# EPICS alarm handler configuration: mps_database/bareTest/alarms/areas/mpln_bpn19_mp01.alhConfig
GROUP NULL MPLN:BPN19:MP01:1
$ALIAS MPS Link Node 83
$GUIDANCE
LTUH MPS
   Group Name: MPLN:BPN19:MP01:1
   Summary PV:  MPLN:BPN19:MP01:1:STATSUMY
$END
CHANNEL  MPLN:BPN19:MP01:1    MPLN:BPN19:MP01:1:MPS_EN_RBV		-----
CHANNEL  MPLN:BPN19:MP01:1    MPLN:BPN19:MP01:1:LC1_MODE_RBV		-----
